(*~
<docu>
	<summary>
		`TcoCarousel` settings/config structure.								
	</summary>				
</docu>	
~*)
TYPE
    TcoCarouselConfig :
    STRUCT

        Direction   : eTcoCarouselDirection;
  		InfoTime : TIME := T#2S;
        ErrorTime : TIME := T#5S;
		NumberOfPositions:UINT;
		// Offset in respect to frist position.
		Offset : UINT;
   
		
    END_STRUCT
END_TYPE

(* stored: Version 1.1.0.1
   DUT TcoCarouselConfig: Id {f96f60b9-8cdd-0314-0d00-7301f489fa2d} *)
